FUNCTION_BLOCK POU
VAR_INPUT
END_VAR
VAR_OUTPUT
END_VAR
VAR
END_VAR

END_FUNCTION_BLOCK

(* stored: Version 1.1.0.1
   POU POU: Id {25e5a927-3f6c-0df0-3967-71e66a9b98ea}, SpecialFunc None *)
